// TIA Portal V20 export
DATA_BLOCK "InstChecksum"   // DB50
AUTHOR : SICAR
FAMILY : Diag
// stored: AssignedProDiagFB ProDiag, InstanceOfName LAF_Checksum, InstanceOfType FB
"LAF_Checksum"
   // VAR_INPUT
   //    plantIdentifier { ExternalAccessible := 'False'; ExternalVisible := 'False'; ExternalWritable := 'False'} : WString[24] := WSTRING#'PLC-Checksum';
   //    textListId { ExternalAccessible := 'False'; ExternalVisible := 'False'; ExternalWritable := 'False'} : Int := 584;
   //    dateTime { ExternalAccessible := 'False'; ExternalVisible := 'False'; ExternalWritable := 'False'} : Date_And_Time := DT#2026-01-06-19:57:41.039;
   //    readChecksum { ExternalAccessible := 'False'; ExternalVisible := 'False'; ExternalWritable := 'False'} : Bool := TRUE;
   //    ack { ExternalAccessible := 'False'; ExternalVisible := 'False'; ExternalWritable := 'False'} : Bool := FALSE;
   //    hideMessageStandard { ExternalAccessible := 'False'; ExternalVisible := 'False'; ExternalWritable := 'False'} : Bool := FALSE;
   //    hideMessageSafety { ExternalAccessible := 'False'; ExternalVisible := 'False'; ExternalWritable := 'False'} : Bool := FALSE;
   //    hideMessageTextlist { ExternalAccessible := 'False'; ExternalVisible := 'False'; ExternalWritable := 'False'} : Bool := FALSE;
   // END_VAR
   // VAR_OUTPUT
   //    generalMessage { ExternalAccessible := 'False'; ExternalVisible := 'False'; ExternalWritable := 'False'} : Bool := FALSE;
   // END_VAR
   // VAR_IN_OUT
   //    checksumHmi : "LAF_typeChecksum";
   // END_VAR
   // VAR
   //    statReadChecksumStorage { ExternalAccessible := 'False'; ExternalVisible := 'False'; ExternalWritable := 'False'} : Bool := FALSE;
   //    statChecksumStandard { ExternalAccessible := 'False'; ExternalVisible := 'False'; ExternalWritable := 'False'} : Array[0..7] of Byte;
   //    statChecksumStafety { ExternalAccessible := 'False'; ExternalVisible := 'False'; ExternalWritable := 'False'} : Array[0..7] of Byte;
   //    statChecksumTextlists { ExternalAccessible := 'False'; ExternalVisible := 'False'; ExternalWritable := 'False'} : Array[0..7] of Byte;
   //    statChecksumStandOldNull { ExternalAccessible := 'False'; ExternalVisible := 'False'; ExternalWritable := 'False'} : Bool := FALSE;
   //    statChecksumSafeOldNull { ExternalAccessible := 'False'; ExternalVisible := 'False'; ExternalWritable := 'False'} : Bool := FALSE;
   //    statChecksumTextlOldNull { ExternalAccessible := 'False'; ExternalVisible := 'False'; ExternalWritable := 'False'} : Bool := FALSE;
   //    statChecksumStandDiff { ExternalAccessible := 'False'; ExternalVisible := 'False'; ExternalWritable := 'False'} : Bool := FALSE;
   //    statChecksumSafeDiff { ExternalAccessible := 'False'; ExternalVisible := 'False'; ExternalWritable := 'False'} : Bool := FALSE;
   //    statChecksumTextlDiff { ExternalAccessible := 'False'; ExternalVisible := 'False'; ExternalWritable := 'False'} : Bool := FALSE;
   //    instGetChecksum1 { ExternalAccessible := 'False'; ExternalVisible := 'False'; ExternalWritable := 'False'} : GetChecksum;
   //    instGetChecksum2 { ExternalAccessible := 'False'; ExternalVisible := 'False'; ExternalWritable := 'False'} : GetChecksum;
   //    instGetChecksum3 { ExternalAccessible := 'False'; ExternalVisible := 'False'; ExternalWritable := 'False'} : GetChecksum;
   //    statRetValHta { ExternalAccessible := 'False'; ExternalVisible := 'False'; ExternalWritable := 'False'} : "LAF_typeChecksumCatWord";
   //    statRisEdgeDiff { ExternalAccessible := 'False'; ExternalVisible := 'False'; ExternalWritable := 'False'} : "LAF_typeChecksumCatBool";
   //    statMessageStandModified { ExternalAccessible := 'False'; ExternalVisible := 'False'; ExternalWritable := 'False'} : Bool := FALSE;
   //    statMessageSafeModified { ExternalAccessible := 'False'; ExternalVisible := 'False'; ExternalWritable := 'False'} : Bool := FALSE;
   //    statMessageTextlModified { ExternalAccessible := 'False'; ExternalVisible := 'False'; ExternalWritable := 'False'} : Bool := FALSE;
   //    statWarnNoStandard { ExternalAccessible := 'False'; ExternalVisible := 'False'; ExternalWritable := 'False'} : UInt := 99;
   //    statWarnNoSafety { ExternalAccessible := 'False'; ExternalVisible := 'False'; ExternalWritable := 'False'} : UInt := 99;
   //    statWarnNoTextlist { ExternalAccessible := 'False'; ExternalVisible := 'False'; ExternalWritable := 'False'} : UInt := 99;
   // END_VAR
BEGIN
   statChecksumStandard[0] := 16#E4;
   statChecksumStandard[1] := 16#AA;
   statChecksumStandard[2] := 16#23;
   statChecksumStandard[3] := 16#DF;
   statChecksumStandard[4] := 16#FD;
   statChecksumStandard[5] := 16#EE;
   statChecksumStandard[6] := 16#A8;
   statChecksumStandard[7] := 16#66;
   statChecksumStafety[0] := 16#0A;
   statChecksumStafety[1] := 16#6C;
   statChecksumStafety[2] := 16#EC;
   statChecksumStafety[3] := 16#4B;
   statChecksumStafety[4..7] := 16#00;
   statChecksumTextlists[0] := 16#67;
   statChecksumTextlists[1] := 16#6D;
   statChecksumTextlists[2] := 16#C4;
   statChecksumTextlists[3] := 16#50;
   statChecksumTextlists[4] := 16#55;
   statChecksumTextlists[5] := 16#90;
   statChecksumTextlists[6] := 16#21;
   statChecksumTextlists[7] := 16#79;
   instGetChecksum1.Scope := 1;
   instGetChecksum1.Done := TRUE;
   instGetChecksum1.Busy := FALSE;
   instGetChecksum1.Error := FALSE;
   instGetChecksum1.Status := 16#0000;
   instGetChecksum1.tmpNulled[0] := 16#E4;
   instGetChecksum1.tmpNulled[1] := 16#AA;
   instGetChecksum1.tmpNulled[2] := 16#23;
   instGetChecksum1.tmpNulled[3] := 16#DF;
   instGetChecksum1.tmpNulled[4] := 16#FD;
   instGetChecksum1.tmpNulled[5] := 16#EE;
   instGetChecksum1.tmpNulled[6] := 16#A8;
   instGetChecksum1.tmpNulled[7] := 16#66;
   instGetChecksum1.GMACount := 1;
   instGetChecksum1.GMAPathLens[0] := 3;
   instGetChecksum1.GMAPaths[0] := 16#89A0_0003;
   instGetChecksum1.GMAPaths[1] := 16#0000_1FC9;
   instGetChecksum1.GMAPaths[2] := 16#0000_0001;
   instGetChecksum1.GMAResLens[0] := 8;
   instGetChecksum2.Scope := 2;
   instGetChecksum2.Done := TRUE;
   instGetChecksum2.Busy := FALSE;
   instGetChecksum2.Error := FALSE;
   instGetChecksum2.Status := 16#0000;
   instGetChecksum2.tmpNulled[0] := 16#0A;
   instGetChecksum2.tmpNulled[1] := 16#6C;
   instGetChecksum2.tmpNulled[2] := 16#EC;
   instGetChecksum2.tmpNulled[3] := 16#4B;
   instGetChecksum2.tmpNulled[4..7] := 16#00;
   instGetChecksum2.GMACount := 1;
   instGetChecksum2.GMAPathLens[0] := 2;
   instGetChecksum2.GMAPaths[0] := 16#89F9_0000;
   instGetChecksum2.GMAPaths[1] := 16#0000_1E37;
   instGetChecksum2.GMAPaths[2] := 16#0000_0000;
   instGetChecksum2.GMAResLens[0] := 4;
   instGetChecksum3.Scope := 3;
   instGetChecksum3.Done := TRUE;
   instGetChecksum3.Busy := FALSE;
   instGetChecksum3.Error := FALSE;
   instGetChecksum3.Status := 16#0000;
   instGetChecksum3.tmpNulled[0] := 16#67;
   instGetChecksum3.tmpNulled[1] := 16#6D;
   instGetChecksum3.tmpNulled[2] := 16#C4;
   instGetChecksum3.tmpNulled[3] := 16#50;
   instGetChecksum3.tmpNulled[4] := 16#55;
   instGetChecksum3.tmpNulled[5] := 16#90;
   instGetChecksum3.tmpNulled[6] := 16#21;
   instGetChecksum3.tmpNulled[7] := 16#79;
   instGetChecksum3.GMACount := 1;
   instGetChecksum3.GMAPathLens[0] := 3;
   instGetChecksum3.GMAPaths[0] := 16#89A0_0072;
   instGetChecksum3.GMAPaths[1] := 16#0000_1FC9;
   instGetChecksum3.GMAPaths[2] := 16#0000_0001;
   instGetChecksum3.GMAResLens[0] := 8;
   statRetValHta.standard := 16#0000;
   statRetValHta.safety := 16#0000;
   statRetValHta.textlists := 16#0000;
   statRisEdgeDiff.standard := FALSE;
   statRisEdgeDiff.safety := FALSE;
   statRisEdgeDiff.textlists := FALSE;
END_DATA_BLOCK
